// TIA Portal V17 export
// export: Created 2021-12-03T08:13:07.5749001Z, ExportSetting WithDefaults, DisplayName Totally Integrated Automation Portal, DisplayVersion V17, DisplayName TIA Portal Openness, DisplayVersion V17, DisplayName TIA Portal Version Control Interface, DisplayVersion V17, DisplayName STEP 7 Professional, DisplayVersion V17, DisplayName STEP 7 Safety, DisplayVersion V17, DisplayName WinCC Advanced, DisplayVersion V17
DATA_BLOCK "DBI_Simulation"   // DB20
VERSION : 0.1
// stored: AutoNumber false, InstanceOfName FB_Simulation, InstanceOfType FB
"FB_Simulation"
BEGIN
END_DATA_BLOCK
